{attribute 'qualified_only'}
// {attribute 'strict'}
TYPE E_FilterOrder :
(
	eFirst := 0,
	eSecond
);
END_TYPE

(* stored: Version 1.1.0.1, ProductVersion 3.1.4024.3
   DUT E_FilterOrder: Id {e81352ad-9a88-46a5-ba1d-363e0f5670da} *)
